FUNCTION_BLOCK Rinstrum_2_AI (* Service Interface Function Block Type *)
  (* Function: All Inputs; Description: Copyright (c) 2018, 2023 Jose Cabral, HR Agrartechnik GmbH This program and the accompanying materials are made available under the terms of the Eclipse Public License 2.0 which is available at https://www.eclipse.org/legal/epl-2.0/ SPDX-License-Identifier: EPL-2.0 this maps to IX *)
  (* Version 1.0, 2018-12-05, Jose Cabral *)
  (* Version 1.1, 2022-08-04, Franz Höpfinger, HR Agrartechnik GmbH *)
  (* Version 1.2, 2023-01-05, Franz Höpfinger, HR Agrartechnik GmbH *)
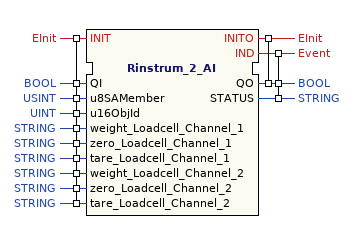
  EVENT_INPUT
    INIT : EInit WITH QI, u8SAMember, u16ObjId, weight_Loadcell_Channel_1, zero_Loadcell_Channel_1, tare_Loadcell_Channel_1, weight_Loadcell_Channel_2, zero_Loadcell_Channel_2, tare_Loadcell_Channel_2; (* Service Initialization *)
  END_EVENT
  EVENT_OUTPUT
    INITO : EInit WITH QO; (* Initialization Confirm *)
    IND WITH QO, STATUS; (* Indication from Resource *)
  END_EVENT
  VAR_INPUT
    QI : BOOL; (* Event Input Qualifier *)
    u8SAMember : USINT := GLOBAL; (* Dummy !, set to GLOBAL if in doubt. OFF deactivates FB. *)
    u16ObjId : UINT := ID_NULL; (* Dummy ! set to ID_NULL if in Doubt. ID_OFF deactivates FB. *)
    weight_Loadcell_Channel_1 : STRING; (* Identifier for Loadcell Channel 1 *)
    zero_Loadcell_Channel_1 : STRING;
    tare_Loadcell_Channel_1 : STRING;
    weight_Loadcell_Channel_2 : STRING; (* Identifier for Loadcell Channel 2 *)
    zero_Loadcell_Channel_2 : STRING;
    tare_Loadcell_Channel_2 : STRING;
  END_VAR
  VAR_OUTPUT
    QO : BOOL; (* Event Output Qualifier *)
    STATUS : STRING; (* Service Status *)
  END_VAR
END_FUNCTION_BLOCK
